PROGRAM PRG_PID_Abwickler
VAR
	Fehler_Abwickler: LREAL;
	eMode							: E_CTRL_MODE;
	stCTRL_P_PARAMS_Abwickler					: ST_CTRL_P_PARAMS;
	stCTRL_I_PARAMS_Abwickler					: ST_CTRL_I_PARAMS;
	stCTRL_D_PARAMS_Abwickler					: ST_CTRL_D_PARAMS;
	eErrorId						: E_CTRL_ERRORCODES;
	bInit							: BOOL	:= TRUE;
	fManSyncValue					: LREAL;
	bSync							: BOOL;
	bError							: BOOL;
	FB_P_Abwickler: FB_CTRL_P;
	FB_I_Abwickler: FB_CTRL_I;
	FB_D_Abwickler: FB_CTRL_D;
	I_Saturation_Abwickler: BOOL;
	PID_Regler_Output_Abwickler: LREAL;
END_VAR

Fehler_Abwickler := Referenzposition - Fadenzugmotor.NcToPlc.ActPos;

IF bInit THEN
	(* init parameter struct *)
	stCTRL_P_PARAMS_Abwickler.tCtrlCycleTime := T#1MS;
	stCTRL_P_PARAMS_Abwickler.tTaskCycleTime := T#1MS;
	stCTRL_P_PARAMS_Abwickler.fKp			 := 1;
	
	stCTRL_I_PARAMS_Abwickler.tCtrlCycleTime := T#100MS;
	stCTRL_I_PARAMS_Abwickler.tTaskCycleTime := T#100MS;
	stCTRL_I_PARAMS_Abwickler.tTi			 := T#50MS;
	stCTRL_I_PARAMS_Abwickler.fOutMaxLimit	 := 40;
	stCTRL_I_PARAMS_Abwickler.fOutMinLimit	 := -40;
	
	stCTRL_D_PARAMS_Abwickler.tCtrlCycleTime := T#1MS;
	stCTRL_D_PARAMS_Abwickler.tTaskCycleTime := T#1MS;
	stCTRL_D_PARAMS_Abwickler.tTv			 := T#3S;
	stCTRL_D_PARAMS_Abwickler.tTd			 := T#10MS;
	stCTRL_D_PARAMS_Abwickler.fOutMaxLimit	 :=  40;
	stCTRL_D_PARAMS_Abwickler.fOutMinLimit	 := -40;

	(* reset the init flag *)
	bInit	:= FALSE;
END_IF	 

(* ein idealer PID-Regler in der Summendarstellung der Parameter *)
FB_PID_Regler_Abwickler();
PID_Regler_Output_Abwickler := P_Regler_Out_Abwickler + I_Regler_Out_Abwickler + D_Regler_Out_Abwickler;	 
//PID_Regler_Output_Abwickler := I_Regler_Out_Abwickler;

IF PID_Regler_Output_Abwickler > 40 THEN 
	PID_Output_After_Saturation_Abwickler := 40;
ELSIF PID_Regler_Output_Abwickler < -40 THEN 
	PID_Output_After_Saturation_Abwickler := -40;
ELSE 
	PID_Output_After_Saturation_Abwickler := PID_Regler_Output_Abwickler;
END_IF	

(* Conditional Intrgration *)
IF Sign(Fehler_Abwickler) = Sign(PID_Regler_Output_Abwickler) AND PID_Output_After_Saturation_Abwickler <> PID_Regler_Output_Abwickler THEN 
	FB_I_Abwickler.bHold := TRUE;
ELSE FB_I_Abwickler.bHold := FALSE;
END_IF

(* Die Richtung der Tänzerregelung anpassen *)
PID_Output_After_Saturation_Abwickler := -PID_Output_After_Saturation_Abwickler;

ACTION FB_PID_Regler_Abwickler:
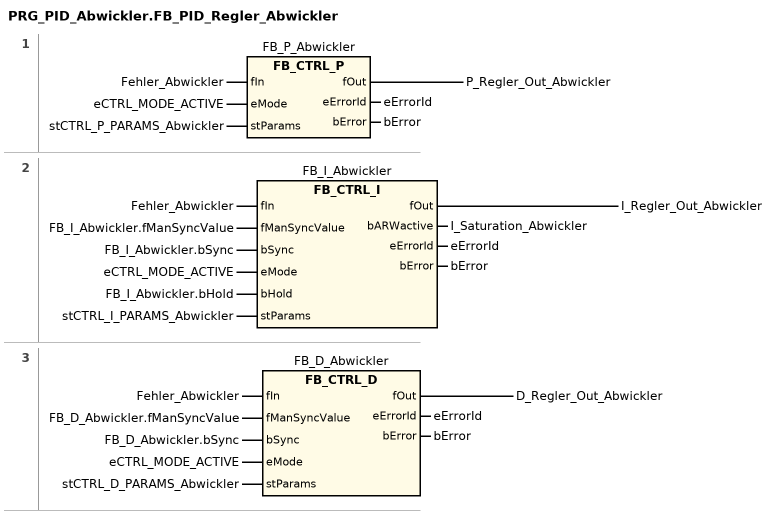
// NETWORK 1
FB_P_Abwickler(
    fIn := Fehler_Abwickler,
    eMode := eCTRL_MODE_ACTIVE,
    stParams := stCTRL_P_PARAMS_Abwickler,
    eErrorId => eErrorId,
    bError => bError); // FB_CTRL_P
P_Regler_Out_Abwickler := FB_P_Abwickler.fOut;

// NETWORK 2
FB_I_Abwickler(
    fIn := Fehler_Abwickler,
    fManSyncValue := FB_I_Abwickler.fManSyncValue,
    bSync := FB_I_Abwickler.bSync,
    eMode := eCTRL_MODE_ACTIVE,
    bHold := FB_I_Abwickler.bHold,
    stParams := stCTRL_I_PARAMS_Abwickler,
    bARWactive => I_Saturation_Abwickler,
    eErrorId => eErrorId,
    bError => bError); // FB_CTRL_I
I_Regler_Out_Abwickler := FB_I_Abwickler.fOut;

// NETWORK 3
FB_D_Abwickler(
    fIn := Fehler_Abwickler,
    fManSyncValue := FB_D_Abwickler.fManSyncValue,
    bSync := FB_D_Abwickler.bSync,
    eMode := eCTRL_MODE_ACTIVE,
    stParams := stCTRL_D_PARAMS_Abwickler,
    eErrorId => eErrorId,
    bError => bError); // FB_CTRL_D
D_Regler_Out_Abwickler := FB_D_Abwickler.fOut;
END_ACTION

END_PROGRAM

(* stored: Version 1.1.0.1, ProductVersion 3.1.4024.11
   POU PRG_PID_Abwickler: Id {1f992af8-526e-4ece-b329-1b1104bc4577}, SpecialFunc None
   Action FB_PID_Regler_Abwickler: Id {c3eb5443-681c-4f6d-b5f8-d0ff4975cf64} *)
